FUNCTION_BLOCK FB_MotionDrive_Test EXTENDS FB_TestSuite
VAR
	stMotionCommand : ST_MotionCommand;
    stMotionStatus: ST_MotionStatus;
	stExMotionStatus : ST_ExtendedMotionStatus;
    fbAxis         : FB_MotionAxisNC_TestDouble;        
    fbInterlocks   : FB_MotionInterlocksLimSw_TestDouble;  
    fbLogger       : FB_MotionLogger_TestDouble;      
    fbMoveRequest  : FB_MoveRequest_TestDouble;        
    fbStateMachine : FB_StateMachine_TestDouble;      
    fbBrake        : FB_Brake_TestDouble;              
END_VAR

NoCrashTest();

METHOD PRIVATE NoCrashTest
VAR_INST
	fbMotionDrive : FB_MotionDrive(	
		stMotionCommand :=stMotionCommand,
		stMotionStatus:=stMotionStatus,
		stExMotionStatus :=stExMotionStatus,
		iInterlocks :=fbInterlocks,
		iLogger :=fbLogger,
		iAxis:=fbAxis,
		iMoveRequest :=fbMoveRequest,
		iStateMachine :=fbStateMachine,
		iBrake :=fbBrake
	);


END_VAR
(*This method is called cyclicly in the fbMotionDrive *)
TEST(__POUNAME());
fbMotionDrive();
TEST_FINISHED();
END_METHOD

END_FUNCTION_BLOCK

(* stored: Version 1.1.0.1
   POU FB_MotionDrive_Test: Id {fa0c0ca3-2ef2-4761-b316-41cf1af95b88}, SpecialFunc None
   Method NoCrashTest: Id {75361fae-01d6-457b-bd6b-fe3e29169e9e} *)
